# EPICS autosave request: iocBoot/ioczzz/APMenu.req
file configMenu.req P=$(P),CONFIG=$(CONFIG)
file analogProc_settings.req  P=$(P),H=$(H)
